(* PLC project  *)

PROGRAM VendorEdgeCases
  VAR
    A : INT;
  END_VAR

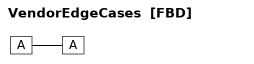
(* FBD diagram, written out as Structured Text *)
A := A;
END_PROGRAM
